FUNCTION_BLOCK TestBoolAdapter2 (* Template for an empty basic function block *)
  (* Standard: 61499-2; Description: Copyright (c) 2019 Jan Holzweber This program and the accompanying materials are made available under the terms of the Eclipse Public License 2.0 which is available at https://www.eclipse.org/legal/epl-2.0/ SPDX-License-Identifier: EPL-2.0 *)
  (* Version 1.0, 2019-07-18, Jan Holzweber *)
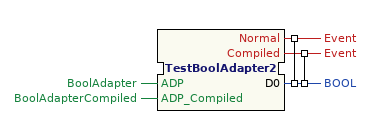
  EVENT_OUTPUT
    Normal WITH D0;
    Compiled WITH D0;
  END_EVENT
  VAR_OUTPUT
    D0 : BOOL;
  END_VAR
  SOCKETS
    ADP : BoolAdapter;
    ADP_Compiled : BoolAdapterCompiled;
  END_SOCKETS
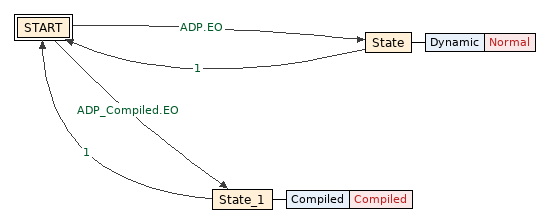
  EC_STATES
    START; (* Initial State *)
    State : Dynamic -> Normal;
    State_1 : Compiled -> Compiled;
  END_STATES
  EC_TRANSITIONS
    START TO State := ADP.EO;
    State TO START := 1;
    START TO State_1 := ADP_Compiled.EO;
    State_1 TO START := 1;
  END_TRANSITIONS
  ALGORITHM Dynamic IN ST: (* new algorithm *)
D0 := ADP.BO;
  END_ALGORITHM
  ALGORITHM Compiled IN ST: (* new algorithm *)
D0 := ADP_Compiled.BO;
  END_ALGORITHM
END_FUNCTION_BLOCK
